(*

## Short summary

This class provides assert statements for floatings (``REAL`` and ``LREAL``)
For 32 bit floats (``REAL``) use `FloatAssertions.single`
For 64 bit floats (``LREAL``) use `FloatAssertions.double`

.. <legal notes>

legal notes
=================
| SPDX-FileCopyrightText: © 2022 ekvip automation GmbH <info@ekvip.de>
| SPDX-License-Identifier: Apache-2.0
| For details check: Apache-2.0_

.. _Apache-2.0: https://www.apache.org/licenses/LICENSE-2.0

.. </legal notes>



*)

{attribute 'reflection'}
FUNCTION_BLOCK INTERNAL FloatAssertions EXTENDS CNM_AbstractObject.Object IMPLEMENTS IFloatAssertions, IAssertCallBacksetter
VAR
	(* class to handle assert statements for 32 bit floats *)
	realAssertions	:RealAssertions();
	(* class to handle assert statements for 64 bit floats *)
	lRealAssertions	:LrealAssertions();
END_VAR

(*

## Short summary
This abstract property returns the class name of the concrete object, 
It's for debugging purpose

.. <legal notes>

legal notes
=================
| SPDX-FileCopyrightText: © 2022 ekvip automation GmbH <info@ekvip.de>
| SPDX-License-Identifier: Apache-2.0
| For details check: Apache-2.0_

.. _Apache-2.0: https://www.apache.org/licenses/LICENSE-2.0

.. </legal notes>

*)

PROPERTY className :CNM_AbstractObject.ClassName
GET
className := 'CNM_Assertor.FloatAssertions';
END_GET
END_PROPERTY

(*

## Short summary
Returns the interface `ILrealAssertions` with assert statements for 64 bit floatings (``LREAL``)

.. <legal notes>

legal notes
=================
| SPDX-FileCopyrightText: © 2022 ekvip automation GmbH <info@ekvip.de>
| SPDX-License-Identifier: Apache-2.0
| For details check: Apache-2.0_

.. _Apache-2.0: https://www.apache.org/licenses/LICENSE-2.0

.. </legal notes>

*)

PROPERTY double :ILrealAssertions
GET
double := THIS^.lRealAssertions;
END_GET
END_PROPERTY

(*

## Short summary
This methods is the setter for the callback class if an assertion was false

.. <legal notes>

legal notes
=================
| SPDX-FileCopyrightText: © 2022 ekvip automation GmbH <info@ekvip.de>
| SPDX-License-Identifier: Apache-2.0
| For details check: Apache-2.0_

.. _Apache-2.0: https://www.apache.org/licenses/LICENSE-2.0

.. </legal notes>



*)

METHOD setCallBack
VAR_INPUT
	(* the class that must be informed if an assertion is false *)
	callBack	:IAssertCallBack;  
END_VAR
THIS^.realAssertions.setCallBack(callBack);
THIS^.lRealAssertions.setCallBack(callBack);
END_METHOD

(*

## Short summary
Returns the interface `IRealAssertions` with assert statements for 32 bit floatings (``REAL``)

.. <legal notes>

legal notes
=================
| SPDX-FileCopyrightText: © 2022 ekvip automation GmbH <info@ekvip.de>
| SPDX-License-Identifier: Apache-2.0
| For details check: Apache-2.0_

.. _Apache-2.0: https://www.apache.org/licenses/LICENSE-2.0

.. </legal notes>

*)

PROPERTY single :IRealAssertions
GET
single := THIS^.realAssertions;
END_GET
END_PROPERTY

END_FUNCTION_BLOCK

(* stored: Version 1.1.0.1, ProductVersion 3.1.4026.12
   POU FloatAssertions: Id {6f765fb2-52a4-4a47-8cd7-95a9639a21cd}, SpecialFunc None
   Property className: Id {bce5ed82-c66d-4d67-b4a1-d5fbfdaf6587}
   Get Get: Id {986d6348-093c-44a4-a3cd-96de1518be0a}
   Property double: Id {05de71a9-9a57-4df4-8c4c-378583055d17}
   Get Get: Id {d020fb99-ff2c-42ee-84be-05cbd018d38d}
   Method setCallBack: Id {9709eb1f-8e3f-403d-a41a-b1be19956e61}
   Property single: Id {2a735a7e-95c4-491b-8de1-8ac0c930d87b}
   Get Get: Id {634a4618-7cca-4f01-bd96-9452c8c3bfec} *)
